{attribute addProperty BoxType "AMP8000-0000-0103-0103"}
{attribute addProperty Id "DeviceDevice_F82A60211620Ch_ACh_A_B17182A2176220WcStateAT %I*WcState_F855686C1620InfoDataAT %I*InfoData_F030DC9B200250"}
{attribute addProperty CRC "4187634827"}
{attribute addProperty SizeInBites "408"}
{attribute addProperty SizeInBytes "51"}
TYPE AMP8000_3F1F35B3 :
STRUCT
	{attribute addProperty Name "Device"}
	Device : Device_F82A6021;
	{attribute addProperty Name "Ch_A"}
	Ch_A : Ch_A_B17182A2;
	{attribute addProperty Name "WcState"}
	WcState : WcState_F855686C;
	{attribute addProperty Name "InfoData"}
	InfoData : InfoData_F030DC9B;
END_STRUCT
END_TYPE

(* stored: Version 1.2.0.0, ProductVersion 3.1.4024.9
   DUT AMP8000_3F1F35B3: Id {7035fa0b-beed-4997-9e9a-474255539ccd} *)
